// Mitsubishi GX Works2 project: 0624(슬라이드실린더_자동_상승펄스_센서)   PLC: Q02/Q02H

PROGRAM MAIN
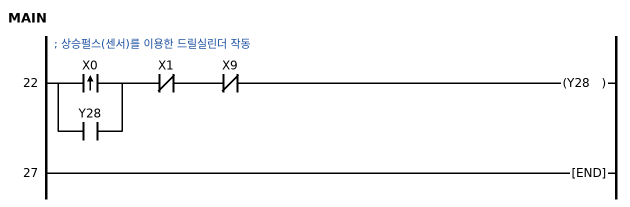
; 상승펄스(센서)를 이용한 드릴실린더 작동
22    LDP     X0
      OR      Y28
      ANI     X1
      ANI     X9
      OUT     Y28
27    END
END_PROGRAM
